// TwinCAT 3 PLC project main
// ProgramVersion: 3.1.4024.0
// libraries:
//   Tc2_Standard, * (Beckhoff Automation GmbH)
//   Tc2_System, * (Beckhoff Automation GmbH)
//   Tc3_Module, * (Beckhoff Automation GmbH)
// project tree:
//   / GlobalTextList.TcGTLO, PlcTask.TcTTO, Visualization Manager.TcVMO (not stored)
//   POUs/ MAIN.TcPOU
//   VISUs/ Visu.TcVIS
// real-time tasks:
//   TASK PlcTask: cycle T#10ms, priority 20, ADS port 350

CONFIGURATION main
    RESOURCE PLC ON TwinCAT3
        TASK PlcTask(INTERVAL := T#10ms, PRIORITY := 20);
        PROGRAM MAIN WITH PlcTask : MAIN;
    END_RESOURCE
END_CONFIGURATION

// ---- POUs/MAIN.TcPOU
PROGRAM MAIN
VAR
	bLamp : BOOL;
	toggle: TON;
	toggleOff: TOF;
END_VAR

toggle(IN:= TRUE, PT:= T#2S , Q=>bLamp , ET=> );
toggleOff(IN:=TRUE , PT:=T#2S , Q=>bLamp , ET=> );

END_PROGRAM

// ---- VISUs/Visu.TcVIS
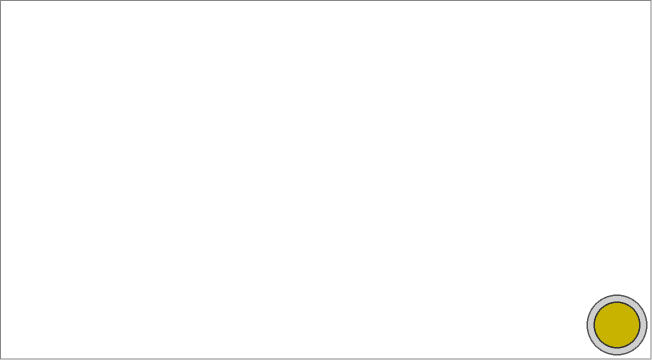
VISUALIZATION Visu  // 652x360
    Lamp1 (582,290 70x70), variable: MAIN.bLamp, style: Lamp-Lamp1-Yellow
END_VISUALIZATION
